// TIA Portal V19 export
VAR_GLOBAL   // PLC tag table "tags_Testtags"
   V1_Test AT %MD30 : Real;
   V2_Test AT %MD34 : Real;
   T1 AT %M38.0 : Bool;
   T2 AT %M38.1 : Bool;
   T3 AT %M38.2 : Bool;
   T4 AT %M38.3 : Bool;
   T5 AT %M38.4 : Bool;
   TI1 AT %MW40 : Int;
   TI2 AT %MW42 : Int;
   TI3 AT %MW44 : Int;
   TI4 AT %MW46 : Int;
END_VAR
